// TIA Portal V19 export
FUNCTION "ALARM" : Void   // FC10, LAD
{ S7_Optimized_Access := 'TRUE' }
// stored: SetENOAutomatically false
   VAR_TEMP   // added for the SCL form of the ladder/FBD networks
      _w1 : Bool;
   END_VAR
BEGIN

REGION Network 1: HOOTER RESET
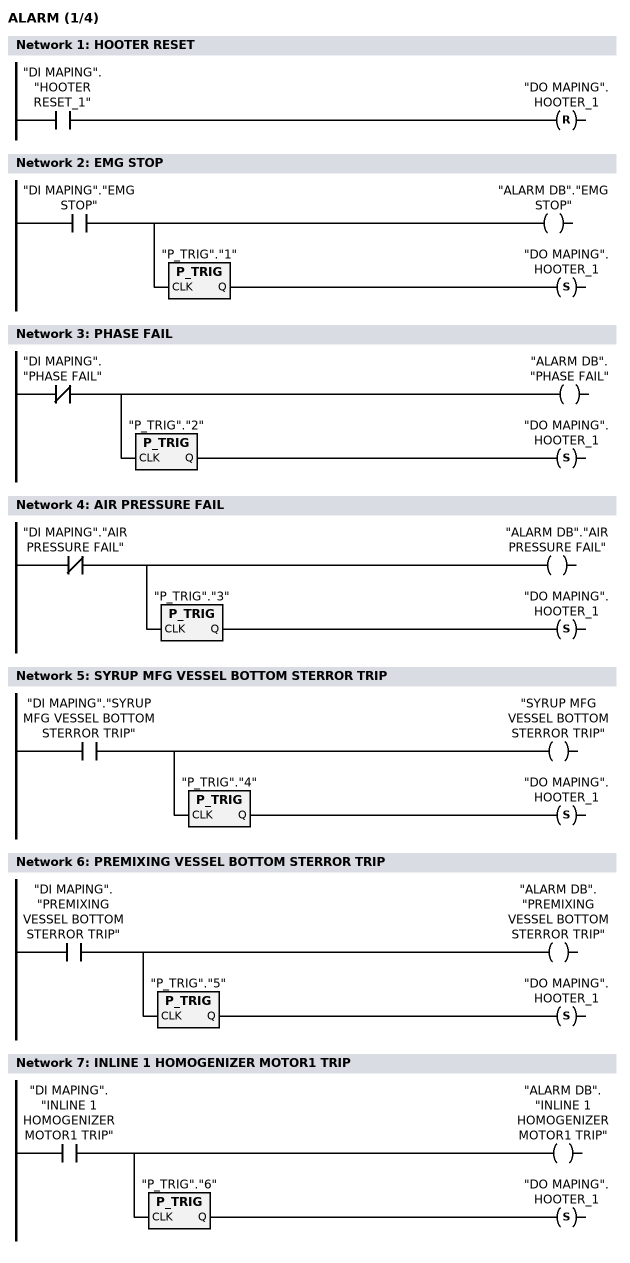
   RUNG wire#powerrail
      Contact( "DI MAPING"."HOOTER RESET_1" )
      R_Coil( "DO MAPING".HOOTER_1 )
   END_RUNG
   // the same network as SCL:
   IF "DI MAPING"."HOOTER RESET_1" THEN "DO MAPING".HOOTER_1 := FALSE; END_IF;
END_REGION

REGION Network 2: EMG STOP
   RUNG wire#powerrail
      Contact( "DI MAPING"."EMG STOP" )
      wire#w1
      Coil( "ALARM DB"."EMG STOP" )
   END_RUNG
   RUNG wire#w1
      P_Trig( "P_TRIG"."1" )
      S_Coil( "DO MAPING".HOOTER_1 )
   END_RUNG
   // the same network as SCL:
   "ALARM DB"."EMG STOP" := "DI MAPING"."EMG STOP";
   #_w1 := "DI MAPING"."EMG STOP" AND NOT "P_TRIG"."1";   // rising edge
   "P_TRIG"."1" := "DI MAPING"."EMG STOP";
   IF #_w1 THEN "DO MAPING".HOOTER_1 := TRUE; END_IF;
END_REGION

REGION Network 3: PHASE FAIL
   RUNG wire#powerrail
      I_Contact( "DI MAPING"."PHASE FAIL" )
      wire#w1
      Coil( "ALARM DB"."PHASE FAIL" )
   END_RUNG
   RUNG wire#w1
      P_Trig( "P_TRIG"."2" )
      S_Coil( "DO MAPING".HOOTER_1 )
   END_RUNG
   // the same network as SCL:
   "ALARM DB"."PHASE FAIL" := NOT "DI MAPING"."PHASE FAIL";
   #_w1 := NOT "DI MAPING"."PHASE FAIL" AND NOT "P_TRIG"."2";   // rising edge
   "P_TRIG"."2" := NOT "DI MAPING"."PHASE FAIL";
   IF #_w1 THEN "DO MAPING".HOOTER_1 := TRUE; END_IF;
END_REGION

REGION Network 4: AIR PRESSURE FAIL
   RUNG wire#powerrail
      I_Contact( "DI MAPING"."AIR PRESSURE FAIL" )
      wire#w1
      Coil( "ALARM DB"."AIR PRESSURE FAIL" )
   END_RUNG
   RUNG wire#w1
      P_Trig( "P_TRIG"."3" )
      S_Coil( "DO MAPING".HOOTER_1 )
   END_RUNG
   // the same network as SCL:
   "ALARM DB"."AIR PRESSURE FAIL" := NOT "DI MAPING"."AIR PRESSURE FAIL";
   #_w1 := NOT "DI MAPING"."AIR PRESSURE FAIL" AND NOT "P_TRIG"."3";   // rising edge
   "P_TRIG"."3" := NOT "DI MAPING"."AIR PRESSURE FAIL";
   IF #_w1 THEN "DO MAPING".HOOTER_1 := TRUE; END_IF;
END_REGION

REGION Network 5: SYRUP MFG VESSEL BOTTOM STERROR TRIP
   RUNG wire#powerrail
      Contact( "DI MAPING"."SYRUP MFG VESSEL BOTTOM STERROR TRIP" )
      wire#w1
      Coil( "SYRUP MFG VESSEL BOTTOM STERROR TRIP" )
   END_RUNG
   RUNG wire#w1
      P_Trig( "P_TRIG"."4" )
      S_Coil( "DO MAPING".HOOTER_1 )
   END_RUNG
   // the same network as SCL:
   "SYRUP MFG VESSEL BOTTOM STERROR TRIP" := "DI MAPING"."SYRUP MFG VESSEL BOTTOM STERROR TRIP";
   #_w1 := "DI MAPING"."SYRUP MFG VESSEL BOTTOM STERROR TRIP" AND NOT "P_TRIG"."4";   // rising edge
   "P_TRIG"."4" := "DI MAPING"."SYRUP MFG VESSEL BOTTOM STERROR TRIP";
   IF #_w1 THEN "DO MAPING".HOOTER_1 := TRUE; END_IF;
END_REGION

REGION Network 6: PREMIXING VESSEL BOTTOM STERROR TRIP
   RUNG wire#powerrail
      Contact( "DI MAPING"."PREMIXING VESSEL BOTTOM STERROR TRIP" )
      wire#w1
      Coil( "ALARM DB"."PREMIXING VESSEL BOTTOM STERROR TRIP" )
   END_RUNG
   RUNG wire#w1
      P_Trig( "P_TRIG"."5" )
      S_Coil( "DO MAPING".HOOTER_1 )
   END_RUNG
   // the same network as SCL:
   "ALARM DB"."PREMIXING VESSEL BOTTOM STERROR TRIP" := "DI MAPING"."PREMIXING VESSEL BOTTOM STERROR TRIP";
   #_w1 := "DI MAPING"."PREMIXING VESSEL BOTTOM STERROR TRIP" AND NOT "P_TRIG"."5";   // rising edge
   "P_TRIG"."5" := "DI MAPING"."PREMIXING VESSEL BOTTOM STERROR TRIP";
   IF #_w1 THEN "DO MAPING".HOOTER_1 := TRUE; END_IF;
END_REGION

REGION Network 7: INLINE 1 HOMOGENIZER MOTOR1 TRIP
   RUNG wire#powerrail
      Contact( "DI MAPING"."INLINE 1 HOMOGENIZER MOTOR1 TRIP" )
      wire#w1
      Coil( "ALARM DB"."INLINE 1 HOMOGENIZER MOTOR1 TRIP" )
   END_RUNG
   RUNG wire#w1
      P_Trig( "P_TRIG"."6" )
      S_Coil( "DO MAPING".HOOTER_1 )
   END_RUNG
   // the same network as SCL:
   "ALARM DB"."INLINE 1 HOMOGENIZER MOTOR1 TRIP" := "DI MAPING"."INLINE 1 HOMOGENIZER MOTOR1 TRIP";
   #_w1 := "DI MAPING"."INLINE 1 HOMOGENIZER MOTOR1 TRIP" AND NOT "P_TRIG"."6";   // rising edge
   "P_TRIG"."6" := "DI MAPING"."INLINE 1 HOMOGENIZER MOTOR1 TRIP";
   IF #_w1 THEN "DO MAPING".HOOTER_1 := TRUE; END_IF;
END_REGION

REGION Network 8: INLINE 2 HOMOGENIZER MOTOR 2 TRIP
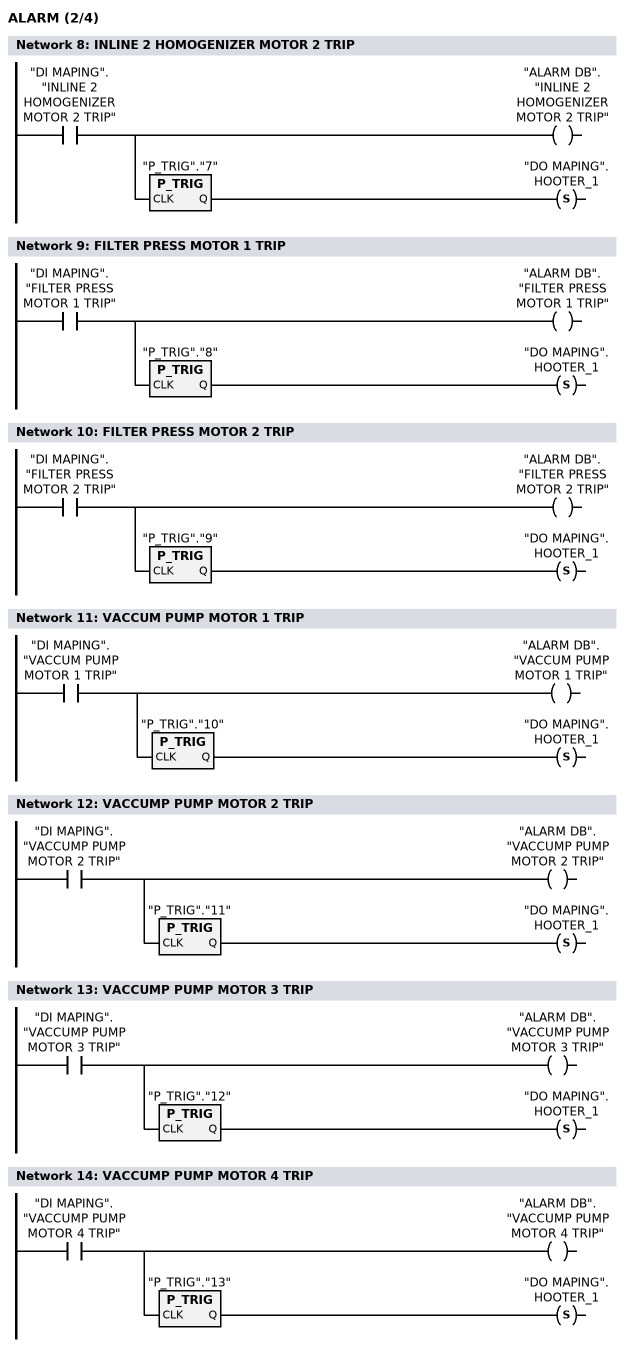
   RUNG wire#powerrail
      Contact( "DI MAPING"."INLINE 2 HOMOGENIZER MOTOR 2 TRIP" )
      wire#w1
      Coil( "ALARM DB"."INLINE 2 HOMOGENIZER MOTOR 2 TRIP" )
   END_RUNG
   RUNG wire#w1
      P_Trig( "P_TRIG"."7" )
      S_Coil( "DO MAPING".HOOTER_1 )
   END_RUNG
   // the same network as SCL:
   "ALARM DB"."INLINE 2 HOMOGENIZER MOTOR 2 TRIP" := "DI MAPING"."INLINE 2 HOMOGENIZER MOTOR 2 TRIP";
   #_w1 := "DI MAPING"."INLINE 2 HOMOGENIZER MOTOR 2 TRIP" AND NOT "P_TRIG"."7";   // rising edge
   "P_TRIG"."7" := "DI MAPING"."INLINE 2 HOMOGENIZER MOTOR 2 TRIP";
   IF #_w1 THEN "DO MAPING".HOOTER_1 := TRUE; END_IF;
END_REGION

REGION Network 9: FILTER PRESS MOTOR 1 TRIP
   RUNG wire#powerrail
      Contact( "DI MAPING"."FILTER PRESS MOTOR 1 TRIP" )
      wire#w1
      Coil( "ALARM DB"."FILTER PRESS MOTOR 1 TRIP" )
   END_RUNG
   RUNG wire#w1
      P_Trig( "P_TRIG"."8" )
      S_Coil( "DO MAPING".HOOTER_1 )
   END_RUNG
   // the same network as SCL:
   "ALARM DB"."FILTER PRESS MOTOR 1 TRIP" := "DI MAPING"."FILTER PRESS MOTOR 1 TRIP";
   #_w1 := "DI MAPING"."FILTER PRESS MOTOR 1 TRIP" AND NOT "P_TRIG"."8";   // rising edge
   "P_TRIG"."8" := "DI MAPING"."FILTER PRESS MOTOR 1 TRIP";
   IF #_w1 THEN "DO MAPING".HOOTER_1 := TRUE; END_IF;
END_REGION

REGION Network 10: FILTER PRESS MOTOR 2 TRIP
   RUNG wire#powerrail
      Contact( "DI MAPING"."FILTER PRESS MOTOR 2 TRIP" )
      wire#w1
      Coil( "ALARM DB"."FILTER PRESS MOTOR 2 TRIP" )
   END_RUNG
   RUNG wire#w1
      P_Trig( "P_TRIG"."9" )
      S_Coil( "DO MAPING".HOOTER_1 )
   END_RUNG
   // the same network as SCL:
   "ALARM DB"."FILTER PRESS MOTOR 2 TRIP" := "DI MAPING"."FILTER PRESS MOTOR 2 TRIP";
   #_w1 := "DI MAPING"."FILTER PRESS MOTOR 2 TRIP" AND NOT "P_TRIG"."9";   // rising edge
   "P_TRIG"."9" := "DI MAPING"."FILTER PRESS MOTOR 2 TRIP";
   IF #_w1 THEN "DO MAPING".HOOTER_1 := TRUE; END_IF;
END_REGION

REGION Network 11: VACCUM PUMP MOTOR 1 TRIP
   RUNG wire#powerrail
      Contact( "DI MAPING"."VACCUM PUMP MOTOR 1 TRIP" )
      wire#w1
      Coil( "ALARM DB"."VACCUM PUMP MOTOR 1 TRIP" )
   END_RUNG
   RUNG wire#w1
      P_Trig( "P_TRIG"."10" )
      S_Coil( "DO MAPING".HOOTER_1 )
   END_RUNG
   // the same network as SCL:
   "ALARM DB"."VACCUM PUMP MOTOR 1 TRIP" := "DI MAPING"."VACCUM PUMP MOTOR 1 TRIP";
   #_w1 := "DI MAPING"."VACCUM PUMP MOTOR 1 TRIP" AND NOT "P_TRIG"."10";   // rising edge
   "P_TRIG"."10" := "DI MAPING"."VACCUM PUMP MOTOR 1 TRIP";
   IF #_w1 THEN "DO MAPING".HOOTER_1 := TRUE; END_IF;
END_REGION

REGION Network 12: VACCUMP PUMP MOTOR 2 TRIP
   RUNG wire#powerrail
      Contact( "DI MAPING"."VACCUMP PUMP MOTOR 2 TRIP" )
      wire#w1
      Coil( "ALARM DB"."VACCUMP PUMP MOTOR 2 TRIP" )
   END_RUNG
   RUNG wire#w1
      P_Trig( "P_TRIG"."11" )
      S_Coil( "DO MAPING".HOOTER_1 )
   END_RUNG
   // the same network as SCL:
   "ALARM DB"."VACCUMP PUMP MOTOR 2 TRIP" := "DI MAPING"."VACCUMP PUMP MOTOR 2 TRIP";
   #_w1 := "DI MAPING"."VACCUMP PUMP MOTOR 2 TRIP" AND NOT "P_TRIG"."11";   // rising edge
   "P_TRIG"."11" := "DI MAPING"."VACCUMP PUMP MOTOR 2 TRIP";
   IF #_w1 THEN "DO MAPING".HOOTER_1 := TRUE; END_IF;
END_REGION

REGION Network 13: VACCUMP PUMP MOTOR 3 TRIP
   RUNG wire#powerrail
      Contact( "DI MAPING"."VACCUMP PUMP MOTOR 3 TRIP" )
      wire#w1
      Coil( "ALARM DB"."VACCUMP PUMP MOTOR 3 TRIP" )
   END_RUNG
   RUNG wire#w1
      P_Trig( "P_TRIG"."12" )
      S_Coil( "DO MAPING".HOOTER_1 )
   END_RUNG
   // the same network as SCL:
   "ALARM DB"."VACCUMP PUMP MOTOR 3 TRIP" := "DI MAPING"."VACCUMP PUMP MOTOR 3 TRIP";
   #_w1 := "DI MAPING"."VACCUMP PUMP MOTOR 3 TRIP" AND NOT "P_TRIG"."12";   // rising edge
   "P_TRIG"."12" := "DI MAPING"."VACCUMP PUMP MOTOR 3 TRIP";
   IF #_w1 THEN "DO MAPING".HOOTER_1 := TRUE; END_IF;
END_REGION

REGION Network 14: VACCUMP PUMP MOTOR 4 TRIP
   RUNG wire#powerrail
      Contact( "DI MAPING"."VACCUMP PUMP MOTOR 4 TRIP" )
      wire#w1
      Coil( "ALARM DB"."VACCUMP PUMP MOTOR 4 TRIP" )
   END_RUNG
   RUNG wire#w1
      P_Trig( "P_TRIG"."13" )
      S_Coil( "DO MAPING".HOOTER_1 )
   END_RUNG
   // the same network as SCL:
   "ALARM DB"."VACCUMP PUMP MOTOR 4 TRIP" := "DI MAPING"."VACCUMP PUMP MOTOR 4 TRIP";
   #_w1 := "DI MAPING"."VACCUMP PUMP MOTOR 4 TRIP" AND NOT "P_TRIG"."13";   // rising edge
   "P_TRIG"."13" := "DI MAPING"."VACCUMP PUMP MOTOR 4 TRIP";
   IF #_w1 THEN "DO MAPING".HOOTER_1 := TRUE; END_IF;
END_REGION

REGION Network 15: SUGAR VESSEL BOTTOM STERROR TRIP
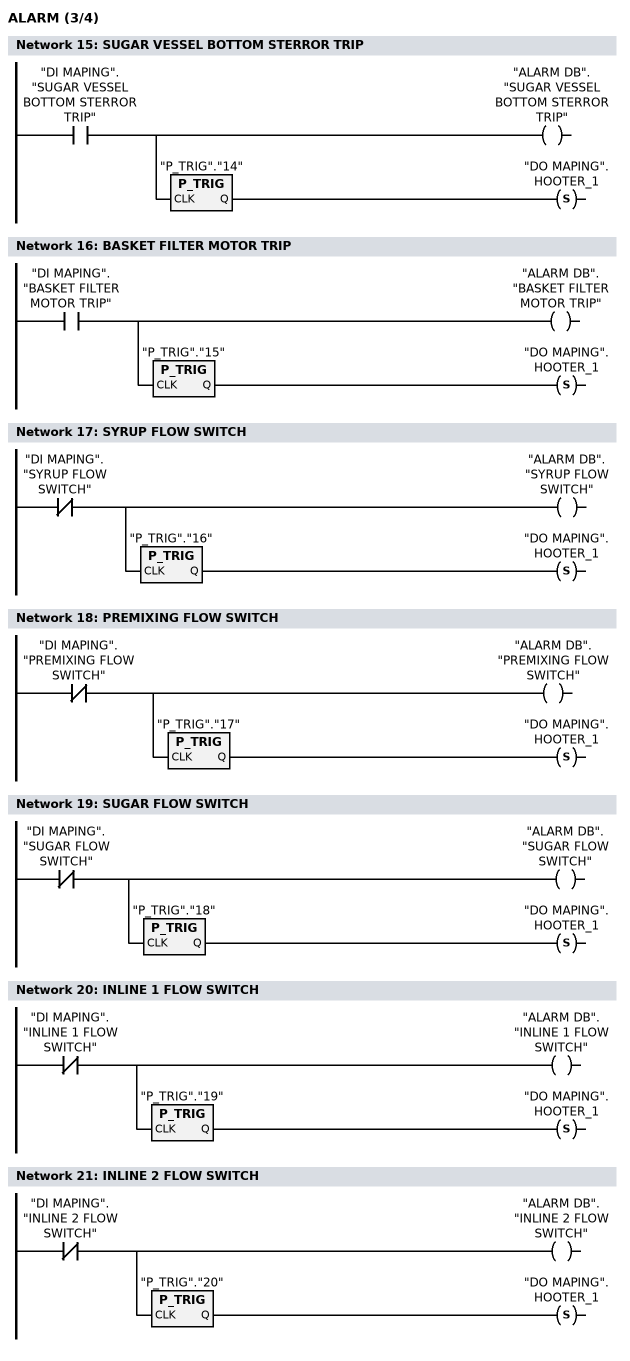
   RUNG wire#powerrail
      Contact( "DI MAPING"."SUGAR VESSEL BOTTOM STERROR TRIP" )
      wire#w1
      Coil( "ALARM DB"."SUGAR VESSEL BOTTOM STERROR TRIP" )
   END_RUNG
   RUNG wire#w1
      P_Trig( "P_TRIG"."14" )
      S_Coil( "DO MAPING".HOOTER_1 )
   END_RUNG
   // the same network as SCL:
   "ALARM DB"."SUGAR VESSEL BOTTOM STERROR TRIP" := "DI MAPING"."SUGAR VESSEL BOTTOM STERROR TRIP";
   #_w1 := "DI MAPING"."SUGAR VESSEL BOTTOM STERROR TRIP" AND NOT "P_TRIG"."14";   // rising edge
   "P_TRIG"."14" := "DI MAPING"."SUGAR VESSEL BOTTOM STERROR TRIP";
   IF #_w1 THEN "DO MAPING".HOOTER_1 := TRUE; END_IF;
END_REGION

REGION Network 16: BASKET FILTER MOTOR TRIP
   RUNG wire#powerrail
      Contact( "DI MAPING"."BASKET FILTER MOTOR TRIP" )
      wire#w1
      Coil( "ALARM DB"."BASKET FILTER MOTOR TRIP" )
   END_RUNG
   RUNG wire#w1
      P_Trig( "P_TRIG"."15" )
      S_Coil( "DO MAPING".HOOTER_1 )
   END_RUNG
   // the same network as SCL:
   "ALARM DB"."BASKET FILTER MOTOR TRIP" := "DI MAPING"."BASKET FILTER MOTOR TRIP";
   #_w1 := "DI MAPING"."BASKET FILTER MOTOR TRIP" AND NOT "P_TRIG"."15";   // rising edge
   "P_TRIG"."15" := "DI MAPING"."BASKET FILTER MOTOR TRIP";
   IF #_w1 THEN "DO MAPING".HOOTER_1 := TRUE; END_IF;
END_REGION

REGION Network 17: SYRUP FLOW SWITCH
   RUNG wire#powerrail
      I_Contact( "DI MAPING"."SYRUP FLOW SWITCH" )
      wire#w1
      Coil( "ALARM DB"."SYRUP FLOW SWITCH" )
   END_RUNG
   RUNG wire#w1
      P_Trig( "P_TRIG"."16" )
      S_Coil( "DO MAPING".HOOTER_1 )
   END_RUNG
   // the same network as SCL:
   "ALARM DB"."SYRUP FLOW SWITCH" := NOT "DI MAPING"."SYRUP FLOW SWITCH";
   #_w1 := NOT "DI MAPING"."SYRUP FLOW SWITCH" AND NOT "P_TRIG"."16";   // rising edge
   "P_TRIG"."16" := NOT "DI MAPING"."SYRUP FLOW SWITCH";
   IF #_w1 THEN "DO MAPING".HOOTER_1 := TRUE; END_IF;
END_REGION

REGION Network 18: PREMIXING FLOW SWITCH
   RUNG wire#powerrail
      I_Contact( "DI MAPING"."PREMIXING FLOW SWITCH" )
      wire#w1
      Coil( "ALARM DB"."PREMIXING FLOW SWITCH" )
   END_RUNG
   RUNG wire#w1
      P_Trig( "P_TRIG"."17" )
      S_Coil( "DO MAPING".HOOTER_1 )
   END_RUNG
   // the same network as SCL:
   "ALARM DB"."PREMIXING FLOW SWITCH" := NOT "DI MAPING"."PREMIXING FLOW SWITCH";
   #_w1 := NOT "DI MAPING"."PREMIXING FLOW SWITCH" AND NOT "P_TRIG"."17";   // rising edge
   "P_TRIG"."17" := NOT "DI MAPING"."PREMIXING FLOW SWITCH";
   IF #_w1 THEN "DO MAPING".HOOTER_1 := TRUE; END_IF;
END_REGION

REGION Network 19: SUGAR FLOW SWITCH
   RUNG wire#powerrail
      I_Contact( "DI MAPING"."SUGAR FLOW SWITCH" )
      wire#w1
      Coil( "ALARM DB"."SUGAR FLOW SWITCH" )
   END_RUNG
   RUNG wire#w1
      P_Trig( "P_TRIG"."18" )
      S_Coil( "DO MAPING".HOOTER_1 )
   END_RUNG
   // the same network as SCL:
   "ALARM DB"."SUGAR FLOW SWITCH" := NOT "DI MAPING"."SUGAR FLOW SWITCH";
   #_w1 := NOT "DI MAPING"."SUGAR FLOW SWITCH" AND NOT "P_TRIG"."18";   // rising edge
   "P_TRIG"."18" := NOT "DI MAPING"."SUGAR FLOW SWITCH";
   IF #_w1 THEN "DO MAPING".HOOTER_1 := TRUE; END_IF;
END_REGION

REGION Network 20: INLINE 1 FLOW SWITCH
   RUNG wire#powerrail
      I_Contact( "DI MAPING"."INLINE 1 FLOW SWITCH" )
      wire#w1
      Coil( "ALARM DB"."INLINE 1 FLOW SWITCH" )
   END_RUNG
   RUNG wire#w1
      P_Trig( "P_TRIG"."19" )
      S_Coil( "DO MAPING".HOOTER_1 )
   END_RUNG
   // the same network as SCL:
   "ALARM DB"."INLINE 1 FLOW SWITCH" := NOT "DI MAPING"."INLINE 1 FLOW SWITCH";
   #_w1 := NOT "DI MAPING"."INLINE 1 FLOW SWITCH" AND NOT "P_TRIG"."19";   // rising edge
   "P_TRIG"."19" := NOT "DI MAPING"."INLINE 1 FLOW SWITCH";
   IF #_w1 THEN "DO MAPING".HOOTER_1 := TRUE; END_IF;
END_REGION

REGION Network 21: INLINE 2 FLOW SWITCH
   RUNG wire#powerrail
      I_Contact( "DI MAPING"."INLINE 2 FLOW SWITCH" )
      wire#w1
      Coil( "ALARM DB"."INLINE 2 FLOW SWITCH" )
   END_RUNG
   RUNG wire#w1
      P_Trig( "P_TRIG"."20" )
      S_Coil( "DO MAPING".HOOTER_1 )
   END_RUNG
   // the same network as SCL:
   "ALARM DB"."INLINE 2 FLOW SWITCH" := NOT "DI MAPING"."INLINE 2 FLOW SWITCH";
   #_w1 := NOT "DI MAPING"."INLINE 2 FLOW SWITCH" AND NOT "P_TRIG"."20";   // rising edge
   "P_TRIG"."20" := NOT "DI MAPING"."INLINE 2 FLOW SWITCH";
   IF #_w1 THEN "DO MAPING".HOOTER_1 := TRUE; END_IF;
END_REGION

REGION Network 22: MFG TO STORAGE-1 WITH INLINE HOMOGENIZER TRANSFER COMPLETE
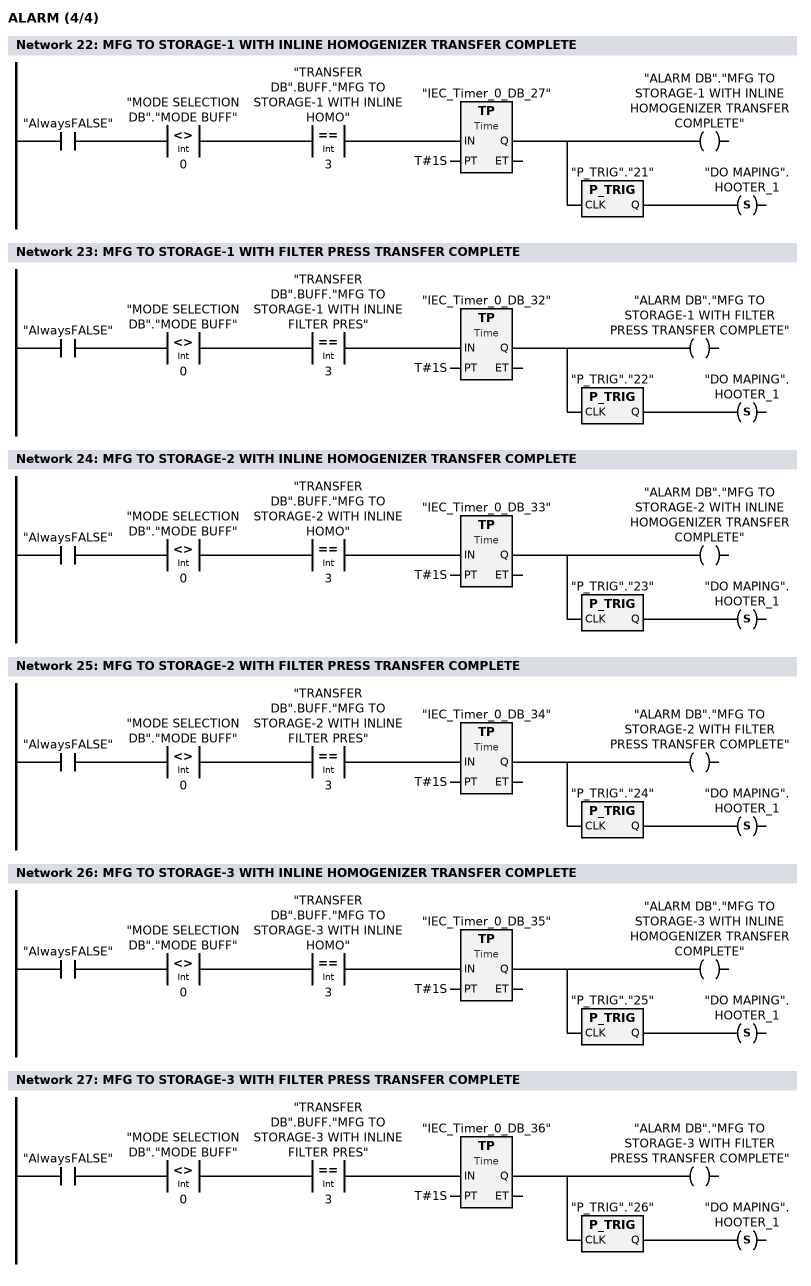
   RUNG wire#powerrail
      Contact( "AlwaysFALSE" )
      { S7_Templates := "SrcType := Int" } NE_Contact(in1 := "MODE SELECTION DB"."MODE BUFF", in2 := 0)
      { S7_Templates := "SrcType := Int" } EQ_Contact(in1 := "TRANSFER DB".BUFF."MFG TO STORAGE-1 WITH INLINE HOMO", in2 := 3)
      { S7_Templates := "time_type := Time" } "IEC_Timer_0_DB_27".TP(pt := T#1S, et =>)
      wire#w1
      Coil( "ALARM DB"."MFG TO STORAGE-1 WITH INLINE HOMOGENIZER TRANSFER COMPLETE" )
   END_RUNG
   RUNG wire#w1
      P_Trig( "P_TRIG"."21" )
      S_Coil( "DO MAPING".HOOTER_1 )
   END_RUNG
   // the same network as SCL:
   "IEC_Timer_0_DB_27".TP(IN := "AlwaysFALSE" AND ("MODE SELECTION DB"."MODE BUFF" <> 0) AND ("TRANSFER DB".BUFF."MFG TO STORAGE-1 WITH INLINE HOMO" = 3),
                          PT := T#1S);
   "ALARM DB"."MFG TO STORAGE-1 WITH INLINE HOMOGENIZER TRANSFER COMPLETE" := "IEC_Timer_0_DB_27".Q;
   #_w1 := "IEC_Timer_0_DB_27".Q AND NOT "P_TRIG"."21";   // rising edge
   "P_TRIG"."21" := "IEC_Timer_0_DB_27".Q;
   IF #_w1 THEN "DO MAPING".HOOTER_1 := TRUE; END_IF;
END_REGION

REGION Network 23: MFG TO STORAGE-1 WITH FILTER PRESS TRANSFER COMPLETE
   RUNG wire#powerrail
      Contact( "AlwaysFALSE" )
      { S7_Templates := "SrcType := Int" } NE_Contact(in1 := "MODE SELECTION DB"."MODE BUFF", in2 := 0)
      { S7_Templates := "SrcType := Int" } EQ_Contact(in1 := "TRANSFER DB".BUFF."MFG TO STORAGE-1 WITH INLINE FILTER PRES", in2 := 3)
      { S7_Templates := "time_type := Time" } "IEC_Timer_0_DB_32".TP(pt := T#1S, et =>)
      wire#w1
      Coil( "ALARM DB"."MFG TO STORAGE-1 WITH FILTER PRESS TRANSFER COMPLETE" )
   END_RUNG
   RUNG wire#w1
      P_Trig( "P_TRIG"."22" )
      S_Coil( "DO MAPING".HOOTER_1 )
   END_RUNG
   // the same network as SCL:
   "IEC_Timer_0_DB_32".TP(IN := "AlwaysFALSE" AND ("MODE SELECTION DB"."MODE BUFF" <> 0) AND ("TRANSFER DB".BUFF."MFG TO STORAGE-1 WITH INLINE FILTER PRES" = 3),
                          PT := T#1S);
   "ALARM DB"."MFG TO STORAGE-1 WITH FILTER PRESS TRANSFER COMPLETE" := "IEC_Timer_0_DB_32".Q;
   #_w1 := "IEC_Timer_0_DB_32".Q AND NOT "P_TRIG"."22";   // rising edge
   "P_TRIG"."22" := "IEC_Timer_0_DB_32".Q;
   IF #_w1 THEN "DO MAPING".HOOTER_1 := TRUE; END_IF;
END_REGION

REGION Network 24: MFG TO STORAGE-2 WITH INLINE HOMOGENIZER TRANSFER COMPLETE
   RUNG wire#powerrail
      Contact( "AlwaysFALSE" )
      { S7_Templates := "SrcType := Int" } NE_Contact(in1 := "MODE SELECTION DB"."MODE BUFF", in2 := 0)
      { S7_Templates := "SrcType := Int" } EQ_Contact(in1 := "TRANSFER DB".BUFF."MFG TO STORAGE-2 WITH INLINE HOMO", in2 := 3)
      { S7_Templates := "time_type := Time" } "IEC_Timer_0_DB_33".TP(pt := T#1S, et =>)
      wire#w1
      Coil( "ALARM DB"."MFG TO STORAGE-2 WITH INLINE HOMOGENIZER TRANSFER COMPLETE" )
   END_RUNG
   RUNG wire#w1
      P_Trig( "P_TRIG"."23" )
      S_Coil( "DO MAPING".HOOTER_1 )
   END_RUNG
   // the same network as SCL:
   "IEC_Timer_0_DB_33".TP(IN := "AlwaysFALSE" AND ("MODE SELECTION DB"."MODE BUFF" <> 0) AND ("TRANSFER DB".BUFF."MFG TO STORAGE-2 WITH INLINE HOMO" = 3),
                          PT := T#1S);
   "ALARM DB"."MFG TO STORAGE-2 WITH INLINE HOMOGENIZER TRANSFER COMPLETE" := "IEC_Timer_0_DB_33".Q;
   #_w1 := "IEC_Timer_0_DB_33".Q AND NOT "P_TRIG"."23";   // rising edge
   "P_TRIG"."23" := "IEC_Timer_0_DB_33".Q;
   IF #_w1 THEN "DO MAPING".HOOTER_1 := TRUE; END_IF;
END_REGION

REGION Network 25: MFG TO STORAGE-2 WITH FILTER PRESS TRANSFER COMPLETE
   RUNG wire#powerrail
      Contact( "AlwaysFALSE" )
      { S7_Templates := "SrcType := Int" } NE_Contact(in1 := "MODE SELECTION DB"."MODE BUFF", in2 := 0)
      { S7_Templates := "SrcType := Int" } EQ_Contact(in1 := "TRANSFER DB".BUFF."MFG TO STORAGE-2 WITH INLINE FILTER PRES", in2 := 3)
      { S7_Templates := "time_type := Time" } "IEC_Timer_0_DB_34".TP(pt := T#1S, et =>)
      wire#w1
      Coil( "ALARM DB"."MFG TO STORAGE-2 WITH FILTER PRESS TRANSFER COMPLETE" )
   END_RUNG
   RUNG wire#w1
      P_Trig( "P_TRIG"."24" )
      S_Coil( "DO MAPING".HOOTER_1 )
   END_RUNG
   // the same network as SCL:
   "IEC_Timer_0_DB_34".TP(IN := "AlwaysFALSE" AND ("MODE SELECTION DB"."MODE BUFF" <> 0) AND ("TRANSFER DB".BUFF."MFG TO STORAGE-2 WITH INLINE FILTER PRES" = 3),
                          PT := T#1S);
   "ALARM DB"."MFG TO STORAGE-2 WITH FILTER PRESS TRANSFER COMPLETE" := "IEC_Timer_0_DB_34".Q;
   #_w1 := "IEC_Timer_0_DB_34".Q AND NOT "P_TRIG"."24";   // rising edge
   "P_TRIG"."24" := "IEC_Timer_0_DB_34".Q;
   IF #_w1 THEN "DO MAPING".HOOTER_1 := TRUE; END_IF;
END_REGION

REGION Network 26: MFG TO STORAGE-3 WITH INLINE HOMOGENIZER TRANSFER COMPLETE
   RUNG wire#powerrail
      Contact( "AlwaysFALSE" )
      { S7_Templates := "SrcType := Int" } NE_Contact(in1 := "MODE SELECTION DB"."MODE BUFF", in2 := 0)
      { S7_Templates := "SrcType := Int" } EQ_Contact(in1 := "TRANSFER DB".BUFF."MFG TO STORAGE-3 WITH INLINE HOMO", in2 := 3)
      { S7_Templates := "time_type := Time" } "IEC_Timer_0_DB_35".TP(pt := T#1S, et =>)
      wire#w1
      Coil( "ALARM DB"."MFG TO STORAGE-3 WITH INLINE HOMOGENIZER TRANSFER COMPLETE" )
   END_RUNG
   RUNG wire#w1
      P_Trig( "P_TRIG"."25" )
      S_Coil( "DO MAPING".HOOTER_1 )
   END_RUNG
   // the same network as SCL:
   "IEC_Timer_0_DB_35".TP(IN := "AlwaysFALSE" AND ("MODE SELECTION DB"."MODE BUFF" <> 0) AND ("TRANSFER DB".BUFF."MFG TO STORAGE-3 WITH INLINE HOMO" = 3),
                          PT := T#1S);
   "ALARM DB"."MFG TO STORAGE-3 WITH INLINE HOMOGENIZER TRANSFER COMPLETE" := "IEC_Timer_0_DB_35".Q;
   #_w1 := "IEC_Timer_0_DB_35".Q AND NOT "P_TRIG"."25";   // rising edge
   "P_TRIG"."25" := "IEC_Timer_0_DB_35".Q;
   IF #_w1 THEN "DO MAPING".HOOTER_1 := TRUE; END_IF;
END_REGION

REGION Network 27: MFG TO STORAGE-3 WITH FILTER PRESS TRANSFER COMPLETE
   RUNG wire#powerrail
      Contact( "AlwaysFALSE" )
      { S7_Templates := "SrcType := Int" } NE_Contact(in1 := "MODE SELECTION DB"."MODE BUFF", in2 := 0)
      { S7_Templates := "SrcType := Int" } EQ_Contact(in1 := "TRANSFER DB".BUFF."MFG TO STORAGE-3 WITH INLINE FILTER PRES", in2 := 3)
      { S7_Templates := "time_type := Time" } "IEC_Timer_0_DB_36".TP(pt := T#1S, et =>)
      wire#w1
      Coil( "ALARM DB"."MFG TO STORAGE-3 WITH FILTER PRESS TRANSFER COMPLETE" )
   END_RUNG
   RUNG wire#w1
      P_Trig( "P_TRIG"."26" )
      S_Coil( "DO MAPING".HOOTER_1 )
   END_RUNG
   // the same network as SCL:
   "IEC_Timer_0_DB_36".TP(IN := "AlwaysFALSE" AND ("MODE SELECTION DB"."MODE BUFF" <> 0) AND ("TRANSFER DB".BUFF."MFG TO STORAGE-3 WITH INLINE FILTER PRES" = 3),
                          PT := T#1S);
   "ALARM DB"."MFG TO STORAGE-3 WITH FILTER PRESS TRANSFER COMPLETE" := "IEC_Timer_0_DB_36".Q;
   #_w1 := "IEC_Timer_0_DB_36".Q AND NOT "P_TRIG"."26";   // rising edge
   "P_TRIG"."26" := "IEC_Timer_0_DB_36".Q;
   IF #_w1 THEN "DO MAPING".HOOTER_1 := TRUE; END_IF;
END_REGION
END_FUNCTION
